# EPICS substitutions: ek9000App/Db/EL4132.substitutions
file EL4132.template
{       pattern
        {
                TERMINAL,

        }
        {
        }
}
